TYPE ST_LaudaWriteCommands_ControlParameters :
STRUCT
	Xp						: STRING := 'OUT_PAR_00_';
	Tn						: STRING := 'OUT_PAR_01_';
	Tv						: STRING := 'OUT_PAR_02_';
	Td						: STRING := 'OUT_PAR_03_';
	KpE						: STRING := 'OUT_PAR_04_';
	TnE						: STRING := 'OUT_PAR_05_';
	TvE						: STRING := 'OUT_PAR_06_';
	TdE						: STRING := 'OUT_PAR_07_';
	CorrectionLimitation	: STRING := 'OUT_PAR_09_';
	XpF						: STRING := 'OUT_PAR_10_';
	Prop_E					: STRING := 'OUT_PAR_15_';
END_STRUCT
END_TYPE

(* stored: Version 1.1.0.1, ProductVersion 3.1.4024.12
   DUT ST_LaudaWriteCommands_ControlParameters: Id {93bff00a-0a65-4884-a882-615ea6707050} *)
